FUNCTION_BLOCK FB_CommandHistory
VAR_OUTPUT
    aCommandHistory: ARRAY [1..nMAX_HISTROY_ENTRY] OF ST_CommandHistoryEntry;
END_VAR
VAR CONSTANT
    nMAX_HISTROY_ENTRY: USINT := 10;
    stEmptyEntry: ST_CommandHistoryEntry := ();
END_VAR

//Shifts the old entries in the history and adds the new command to the top
METHOD mAdd
VAR_INPUT
    eCommand: E_MotionFunctions;
END_VAR
//Shift old entries
IF nMAX_HISTROY_ENTRY > 1 THEN
    MEMMOVE(
        destAddr := ADR(aCommandHistory[2]),
        srcAddr := ADR(aCommandHistory),
        n := (nMAX_HISTROY_ENTRY - 1) * SIZEOF(ST_CommandHistoryEntry));
END_IF

//Clear old entry
aCommandHistory[1] := stEmptyEntry;

//Add new entry
aCommandHistory[1].eCommand := eCommand;
aCommandHistory[1].dtTrigger := FILETIME64_TO_DT(F_GetSystemTime());
END_METHOD

//Sets the release time of the top entry
METHOD mSetRelease
aCommandHistory[1].dtRelease := FILETIME64_TO_DT(F_GetSystemTime());
END_METHOD

END_FUNCTION_BLOCK

(* stored: Version 1.1.0.1
   POU FB_CommandHistory: Id {39e94074-e42b-0657-2248-14d00ab28c33}, SpecialFunc None
   Method mAdd: Id {814dbda4-eaf2-055a-2536-42e29c3098af}
   Method mSetRelease: Id {340a6c28-35e6-0fbc-3027-e0dab46adcda} *)
